FUNCTION_BLOCK Stage14 (* Template for a Basic Function Block Type *)
  (* Standard: 61499-2 *)
  (* Version 1.0, 2021-06-20, HP *)
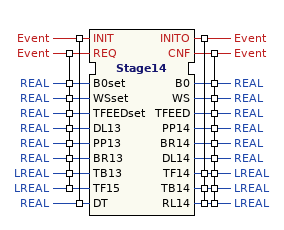
  EVENT_INPUT
    INIT WITH DT; (* Initialization Request *)
    REQ WITH B0set, WSset, TFEEDset, DL13, PP13, BR13, TB13, TF15; (* Normal Execution Request *)
  END_EVENT
  EVENT_OUTPUT
    INITO WITH TB14, RL14, TF14; (* Initialization Confirm *)
    CNF WITH TB14, DL14, TF14, BR14, PP14, B0, WS, TFEED, RL14; (* Execution Confirmation *)
  END_EVENT
  VAR_INPUT
    B0set : REAL;
    WSset : REAL;
    TFEEDset : REAL;
    DL13 : REAL;
    PP13 : REAL;
    BR13 : REAL;
    TB13 : LREAL;
    TF15 : LREAL;
    DT : REAL;
  END_VAR
  VAR_OUTPUT
    B0 : REAL;
    WS : REAL;
    TFEED : REAL;
    PP14 : REAL;
    BR14 : REAL;
    DL14 : REAL;
    TF14 : LREAL;
    TB14 : LREAL;
    RL14 : LREAL;
  END_VAR
  VAR
    AB : REAL; (* internal variabel *)
    UU : REAL;
    TREF : REAL;
    AD : REAL;
    AHC : REAL;
    AHR : REAL;
    AS : REAL;
    REC : REAL;
    WN : REAL;
    WN_1 : REAL;
    XKN : REAL;
    C1 : REAL;
    HS : REAL;
    G : REAL;
    W1 : REAL;
    TFREC : REAL;
    TS : REAL;
    DTS : REAL;
    TF14_last : REAL;
    RL14_last : REAL;
    TB14_last : REAL;
    USS : REAL;
    RHOB : REAL;
    CPB : REAL;
    CPF : REAL;
    FMW : REAL;
    HLV : REAL;
    HV : REAL;
    BPR : REAL;
    FMC : REAL;
    U : REAL;
    A : REAL;
    B : REAL;
    C : REAL;
    D1 : REAL;
    d : REAL;
    a : REAL;
    A1 : REAL;
    A2 : REAL;
    A3 : REAL;
    A4 : REAL;
    A5 : REAL;
    A6 : REAL;
    p : REAL;
    q : REAL;
    TC : REAL;
    PC : REAL;
    DTB14 : REAL;
    DEN14 : REAL;
    DH14 : REAL;
    DP14 : REAL;
    DPDH14 : REAL;
    DT14 : REAL;
    m : REAL;
    n : REAL;
    VR14 : REAL;
    DELTA14 : REAL;
    DELTA36 : REAL;
    DELTA58 : REAL;
    DELTA14_last : REAL;
    DELTA36_last : REAL;
    DELTA58_last : REAL;
  END_VAR
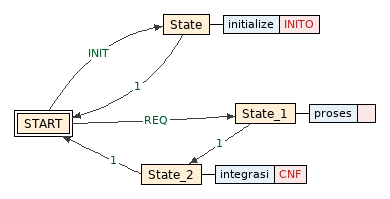
  EC_STATES
    START; (* Initial State *)
    State : initialize -> INITO;
    State_1 : proses;
    State_2 : integrasi -> CNF;
  END_STATES
  EC_TRANSITIONS
    START TO State := INIT;
    State TO START := 1;
    START TO State_1 := REQ;
    State_1 TO State_2 := 1;
    State_2 TO START := 1;
  END_TRANSITIONS
  ALGORITHM initialize IN ST: (* Initialization algorithm *)
TREF :=273.15;
AB :=57.2727;
AHC :=4069.2;
AHR :=2639.7;
AS :=3225.7;
REC :=0.0;
//TF2:=TF2;

//TFEED :=TFEED1+TREF;
 //TS:=TS1+TREF;
WN :=3.0;
XKN :=0.68;
HS:=0.11;
G :=9.81;
W1 :=0.50;

RL14 := 0.598669333203972;
TB14 := 330.414960218012;
TF14 := 326.857347111076;
TF15 := 324.575567486082;



RL14_last :=RL14;
TB14_last :=TB14;
TF14_last :=TF14;
  END_ALGORITHM
  ALGORITHM proses IN ST: (* kalkulasi *)
B0 :=B0set;
WS :=WSset;
TFEED:=TFEEDset;
UU := TFEEDset;
U :=UU;

USS :=49.767;
C1 :=0.625;
RHOB :=1032.4; //maassa jenis brine
CPB :=1.00; //heatcapacity Brine
CPF :=1.00; //heat capacity feed
FMW :=23654.0;
HLV :=563.7959;
HV :=625.1971;
BPR :=2.192;
FMC :=34736.09;
//U :=UU; //feed temp



///  Calculate the physical properties

//A :=3.2437814;
//B :=5.86826*0.001;
//C :=1.1702379*0.00000001;
//D1 :=2.1878462*0.001;
//TC :=647.27;
//PC :=218.167;


A1 :=3.2437814;
A2:=5.86826*0.001;
A3:=1.1702379*0.00000001;
A4 :=2.1878462*0.001;
A5 :=647.27;
A6 :=218.167;

DTB14 :=A5-TB14;
DEN14 :=(A1+A2*DTB14+A3*DTB14*DTB14*DTB14)/(1+A4*DTB14)*DTB14/TB14;
p:=DEN14;
q:=10.0;
PP14 :=A6/(EXPT(q, p));

// calculate the brine flow rates
DP14:=PP13-PP14;
DH14:=RL14-C1*HS;
DPDH14 :=DP14*101000+G*RHOB*DH14;
m:=DPDH14*RHOB;
n:=0.5;
BR14 :=WN*XKN*RL14*(EXPT(m, n));
BR14 :=BR14*60.0/1000.0;

// calculate the vapor flow rates

DT14 :=TB14-BPR/1.8-(TF15+TF14)*0.5;
VR14:=U*AHC*DT14/HLV/1000.0;
DL14 :=DL13+VR14;


//// state equation
DELTA14 :=(BR13-BR14-VR14)*1000.0/RHOB/AB;
DELTA36 :=((BR13*CPB*(TB13-TB14))-VR14*(HV-CPB*(TB14-TREF)))*1000.0/AB/RHOB/CPB/RL14;
DELTA58 :=(B0*CPF*(TF15-TF14)*1000+(U*AHC*DT14))/FMW/CPF;
  END_ALGORITHM
  ALGORITHM integrasi IN ST: (* new algorithm *)
B0 :=B0set;
WS :=WSset;
TFEED := TFEEDset;
//integrasi
RL14 := (DELTA14 + DELTA14_last)*0.5*DT + RL14_last;
DELTA14_last :=DELTA14 ;
RL14_last :=RL14;

TB14:= (DELTA36 + DELTA36_last)*0.5*DT + TB14_last;
DELTA36_last :=DELTA36 ;
TB14_last:=TB14;

TF14 := (DELTA58 + DELTA58_last)*0.5*DT + TF14_last;
DELTA58_last :=DELTA58 ;
TF14_last :=TF14;
  END_ALGORITHM
END_FUNCTION_BLOCK
